{attribute 'GeneratedUsingTerminal: EK1100-0000-0018'}
{attribute addProperty BoxType "EK1100-0000-0018"}
{attribute addProperty Id "Beckhoff_EP4xxxEK1122Beckhoff_EP4xxxEK1122_3C25AF73256"}
{attribute addProperty CRC "433942213"}
{attribute addProperty Size "256"}
TYPE Beckhoff_EP4xxx_19DD6EC5 EXTENDS EK1100_1FC0878B :
STRUCT
	{attribute addProperty Name "Beckhoff_EP4xxxEK1122"}
	{attribute addProperty PreviousPort "Beckhoff EP4xxx : B"}
	Beckhoff_EP4xxxEK1122 : Beckhoff_EP4xxxEK1122_3C25AF73;
END_STRUCT
END_TYPE

(* stored: Version 1.2.0.0, ProductVersion 3.1.4024.9
   DUT Beckhoff_EP4xxx_19DD6EC5: Id {7897593c-2900-4b3b-ba8b-c860b13e8415} *)
